// TwinCAT 3 PLC project Untitled1
// ProgramVersion: 3.1.4023.0
// libraries:
//   OpenWeatherMap, * (Stefan Besler)
//   Tc2_Standard, * (Beckhoff Automation GmbH)
//   Tc2_System, * (Beckhoff Automation GmbH)
//   Tc3_Module, * (Beckhoff Automation GmbH)
// project tree:
//   / PlcTask.TcTTO
//   POUs/ MAIN.TcPOU
// real-time tasks:
//   TASK PlcTask: cycle T#10ms, priority 20, ADS port 350

CONFIGURATION Untitled1
    RESOURCE PLC ON TwinCAT3
        TASK PlcTask(INTERVAL := T#10ms, PRIORITY := 20);
        PROGRAM MAIN WITH PlcTask : MAIN;
    END_RESOURCE
END_CONFIGURATION

// ---- POUs/MAIN.TcPOU
PROGRAM MAIN
VAR
  _send : BOOL; // boolean, which can be triggered to send a message
  _openWeatherMapClient : OpenWeatherMap.OpenWeatherMapClient('<your_token>');   
END_VAR

IF _send
THEN
  _send := FALSE;
  _openWeatherMapClient.RequestWeatherByZipCodeAsync('6020', 'AT');
END_IF

_openWeatherMapClient.Cyclic();

END_PROGRAM
